// TwinCAT 3 PLC project PLC
// ProgramVersion: 3.1.4026.19
// libraries:
//   Tc2_DMX, * (Beckhoff Automation GmbH)
//   Tc2_Standard, * (Beckhoff Automation GmbH)
//   Tc2_System, * (Beckhoff Automation GmbH)
// project tree:
//   DUTs/ ENUM_InternalControl_StateMachine.TcDUT
//   GVLs/ GVL_DMX.TcGVL
//   POUs/ FB_ModuleLEDs.TcPOU, P_TestModuleLEDs.TcPOU
//   / Task.TcTTO
// real-time tasks:
//   TASK Task: cycle T#10ms, priority 1, ADS port 350
// I/O:
//   DEVICE Device 1 (EtherCAT), AmsNetId 10.1.181.84.2.1
//     Term 6 (EK1200) [EK1200-5000 EtherCAT Power supply (2A E-Bus)]
//       Term 3 (EL1809) [EL1809 16Ch. Dig. Input 24V, 3ms]
//       Term 4 (EL1809) [EL1809 16Ch. Dig. Input 24V, 3ms]
//       Term 5 (EL2008) [EL2008 8Ch. Dig. Output 24V, 0.5A]
//       Term 7 (EL2008) [EL2008 8Ch. Dig. Output 24V, 0.5A]
//       Term 8 (EL6851) [EL6851 DMX Master]
//       Term 12 (EL9011) [EL9011 End Terminal]
//   DEVICE Device 4 (USB) (disabled)
//   DEVICE Device 5 (COM Port) (disabled)
// variable links:
//   Device 1 (EtherCAT) <-> Device 1 (EtherCAT)/Term 6 (EK1200)/Term 5 (EL2008)
//     Term 6 (EK1200)/Term 3 (EL1809)/Channel 1/Input <-> Channel 1/Output
//   PLC/PLC Instance <-> Device 1 (EtherCAT)/Term 6 (EK1200)/Term 8 (EL6851)
//     Task Inputs/GVL_DMX.stDMXInDataLine01/bCyclicTxDDisabled <-> DMX Status/Cyclic TxD disabled
//     Task Inputs/GVL_DMX.stDMXInDataLine01/bDefaultDataSent <-> DMX Status/Default data sent
//     Task Inputs/GVL_DMX.stDMXInDataLine01/bFrameSentToggle <-> DMX Status/Frame sent toggle
//     Task Inputs/GVL_DMX.stDMXInDataLine01/bReceiveToggle <-> DMX Status/Receive toggle
//     Task Inputs/GVL_DMX.stDMXInDataLine01/bTransmitAccepted <-> DMX Status/Transmit accepted
//     Task Inputs/GVL_DMX.stDMXInDataLine01/bTxPDOToggle <-> DMX Status/TxPDO Toggle
//     Task Inputs/GVL_DMX.stDMXInDataLine01/byStartCode <-> DMX Status/Start code
//     Task Inputs/GVL_DMX.stDMXInDataLine01/wChannelLength <-> DMX Status/Channel length
//     Task Outputs/GVL_DMX.stDMXOutDataLine01/arrData[100] <-> DMX Channel 65-128/Channel 100
//     Task Outputs/GVL_DMX.stDMXOutDataLine01/arrData[101] <-> DMX Channel 65-128/Channel 101
//     Task Outputs/GVL_DMX.stDMXOutDataLine01/arrData[102] <-> DMX Channel 65-128/Channel 102
//     Task Outputs/GVL_DMX.stDMXOutDataLine01/arrData[103] <-> DMX Channel 65-128/Channel 103
//     Task Outputs/GVL_DMX.stDMXOutDataLine01/arrData[104] <-> DMX Channel 65-128/Channel 104
//     Task Outputs/GVL_DMX.stDMXOutDataLine01/arrData[105] <-> DMX Channel 65-128/Channel 105
//     Task Outputs/GVL_DMX.stDMXOutDataLine01/arrData[106] <-> DMX Channel 65-128/Channel 106
//     Task Outputs/GVL_DMX.stDMXOutDataLine01/arrData[107] <-> DMX Channel 65-128/Channel 107
//     Task Outputs/GVL_DMX.stDMXOutDataLine01/arrData[108] <-> DMX Channel 65-128/Channel 108
//     Task Outputs/GVL_DMX.stDMXOutDataLine01/arrData[109] <-> DMX Channel 65-128/Channel 109
//     Task Outputs/GVL_DMX.stDMXOutDataLine01/arrData[10] <-> DMX Channel 1-64/Channel 10
//     Task Outputs/GVL_DMX.stDMXOutDataLine01/arrData[110] <-> DMX Channel 65-128/Channel 110
//     Task Outputs/GVL_DMX.stDMXOutDataLine01/arrData[111] <-> DMX Channel 65-128/Channel 111
//     Task Outputs/GVL_DMX.stDMXOutDataLine01/arrData[112] <-> DMX Channel 65-128/Channel 112
//     Task Outputs/GVL_DMX.stDMXOutDataLine01/arrData[113] <-> DMX Channel 65-128/Channel 113
//     Task Outputs/GVL_DMX.stDMXOutDataLine01/arrData[114] <-> DMX Channel 65-128/Channel 114
//     Task Outputs/GVL_DMX.stDMXOutDataLine01/arrData[115] <-> DMX Channel 65-128/Channel 115
//     Task Outputs/GVL_DMX.stDMXOutDataLine01/arrData[116] <-> DMX Channel 65-128/Channel 116
//     Task Outputs/GVL_DMX.stDMXOutDataLine01/arrData[117] <-> DMX Channel 65-128/Channel 117
//     Task Outputs/GVL_DMX.stDMXOutDataLine01/arrData[118] <-> DMX Channel 65-128/Channel 118
//     Task Outputs/GVL_DMX.stDMXOutDataLine01/arrData[119] <-> DMX Channel 65-128/Channel 119
//     Task Outputs/GVL_DMX.stDMXOutDataLine01/arrData[11] <-> DMX Channel 1-64/Channel 11
//     Task Outputs/GVL_DMX.stDMXOutDataLine01/arrData[120] <-> DMX Channel 65-128/Channel 120
//     Task Outputs/GVL_DMX.stDMXOutDataLine01/arrData[121] <-> DMX Channel 65-128/Channel 121
//     Task Outputs/GVL_DMX.stDMXOutDataLine01/arrData[122] <-> DMX Channel 65-128/Channel 122
//     Task Outputs/GVL_DMX.stDMXOutDataLine01/arrData[123] <-> DMX Channel 65-128/Channel 123
//     Task Outputs/GVL_DMX.stDMXOutDataLine01/arrData[124] <-> DMX Channel 65-128/Channel 124
//     Task Outputs/GVL_DMX.stDMXOutDataLine01/arrData[125] <-> DMX Channel 65-128/Channel 125
//     Task Outputs/GVL_DMX.stDMXOutDataLine01/arrData[126] <-> DMX Channel 65-128/Channel 126
//     Task Outputs/GVL_DMX.stDMXOutDataLine01/arrData[127] <-> DMX Channel 65-128/Channel 127
//     Task Outputs/GVL_DMX.stDMXOutDataLine01/arrData[128] <-> DMX Channel 65-128/Channel 128
//     Task Outputs/GVL_DMX.stDMXOutDataLine01/arrData[12] <-> DMX Channel 1-64/Channel 12
//     Task Outputs/GVL_DMX.stDMXOutDataLine01/arrData[13] <-> DMX Channel 1-64/Channel 13
//     Task Outputs/GVL_DMX.stDMXOutDataLine01/arrData[14] <-> DMX Channel 1-64/Channel 14
//     Task Outputs/GVL_DMX.stDMXOutDataLine01/arrData[15] <-> DMX Channel 1-64/Channel 15
//     Task Outputs/GVL_DMX.stDMXOutDataLine01/arrData[16] <-> DMX Channel 1-64/Channel 16
//     Task Outputs/GVL_DMX.stDMXOutDataLine01/arrData[17] <-> DMX Channel 1-64/Channel 17
//     Task Outputs/GVL_DMX.stDMXOutDataLine01/arrData[18] <-> DMX Channel 1-64/Channel 18
//     Task Outputs/GVL_DMX.stDMXOutDataLine01/arrData[19] <-> DMX Channel 1-64/Channel 19
//     Task Outputs/GVL_DMX.stDMXOutDataLine01/arrData[1] <-> DMX Channel 1-64/Channel 1
//     Task Outputs/GVL_DMX.stDMXOutDataLine01/arrData[20] <-> DMX Channel 1-64/Channel 20
//     Task Outputs/GVL_DMX.stDMXOutDataLine01/arrData[21] <-> DMX Channel 1-64/Channel 21
//     Task Outputs/GVL_DMX.stDMXOutDataLine01/arrData[22] <-> DMX Channel 1-64/Channel 22
//     Task Outputs/GVL_DMX.stDMXOutDataLine01/arrData[23] <-> DMX Channel 1-64/Channel 23
//     Task Outputs/GVL_DMX.stDMXOutDataLine01/arrData[24] <-> DMX Channel 1-64/Channel 24
//     Task Outputs/GVL_DMX.stDMXOutDataLine01/arrData[25] <-> DMX Channel 1-64/Channel 25
//     Task Outputs/GVL_DMX.stDMXOutDataLine01/arrData[26] <-> DMX Channel 1-64/Channel 26
//     Task Outputs/GVL_DMX.stDMXOutDataLine01/arrData[27] <-> DMX Channel 1-64/Channel 27
//     Task Outputs/GVL_DMX.stDMXOutDataLine01/arrData[28] <-> DMX Channel 1-64/Channel 28
//     Task Outputs/GVL_DMX.stDMXOutDataLine01/arrData[29] <-> DMX Channel 1-64/Channel 29
//     Task Outputs/GVL_DMX.stDMXOutDataLine01/arrData[2] <-> DMX Channel 1-64/Channel 2
//     Task Outputs/GVL_DMX.stDMXOutDataLine01/arrData[30] <-> DMX Channel 1-64/Channel 30
//     Task Outputs/GVL_DMX.stDMXOutDataLine01/arrData[31] <-> DMX Channel 1-64/Channel 31
//     Task Outputs/GVL_DMX.stDMXOutDataLine01/arrData[32] <-> DMX Channel 1-64/Channel 32
//     Task Outputs/GVL_DMX.stDMXOutDataLine01/arrData[33] <-> DMX Channel 1-64/Channel 33
//     Task Outputs/GVL_DMX.stDMXOutDataLine01/arrData[34] <-> DMX Channel 1-64/Channel 34
//     Task Outputs/GVL_DMX.stDMXOutDataLine01/arrData[35] <-> DMX Channel 1-64/Channel 35
//     Task Outputs/GVL_DMX.stDMXOutDataLine01/arrData[36] <-> DMX Channel 1-64/Channel 36
//     Task Outputs/GVL_DMX.stDMXOutDataLine01/arrData[37] <-> DMX Channel 1-64/Channel 37
//     Task Outputs/GVL_DMX.stDMXOutDataLine01/arrData[38] <-> DMX Channel 1-64/Channel 38
//     Task Outputs/GVL_DMX.stDMXOutDataLine01/arrData[39] <-> DMX Channel 1-64/Channel 39
//     Task Outputs/GVL_DMX.stDMXOutDataLine01/arrData[3] <-> DMX Channel 1-64/Channel 3
//     Task Outputs/GVL_DMX.stDMXOutDataLine01/arrData[40] <-> DMX Channel 1-64/Channel 40
//     Task Outputs/GVL_DMX.stDMXOutDataLine01/arrData[41] <-> DMX Channel 1-64/Channel 41
//     Task Outputs/GVL_DMX.stDMXOutDataLine01/arrData[42] <-> DMX Channel 1-64/Channel 42
//     Task Outputs/GVL_DMX.stDMXOutDataLine01/arrData[43] <-> DMX Channel 1-64/Channel 43
//     Task Outputs/GVL_DMX.stDMXOutDataLine01/arrData[44] <-> DMX Channel 1-64/Channel 44
//     Task Outputs/GVL_DMX.stDMXOutDataLine01/arrData[45] <-> DMX Channel 1-64/Channel 45
//     Task Outputs/GVL_DMX.stDMXOutDataLine01/arrData[46] <-> DMX Channel 1-64/Channel 46
//     Task Outputs/GVL_DMX.stDMXOutDataLine01/arrData[47] <-> DMX Channel 1-64/Channel 47
//     Task Outputs/GVL_DMX.stDMXOutDataLine01/arrData[48] <-> DMX Channel 1-64/Channel 48
//     Task Outputs/GVL_DMX.stDMXOutDataLine01/arrData[49] <-> DMX Channel 1-64/Channel 49
//     Task Outputs/GVL_DMX.stDMXOutDataLine01/arrData[4] <-> DMX Channel 1-64/Channel 4
//     Task Outputs/GVL_DMX.stDMXOutDataLine01/arrData[50] <-> DMX Channel 1-64/Channel 50
//     Task Outputs/GVL_DMX.stDMXOutDataLine01/arrData[51] <-> DMX Channel 1-64/Channel 51
//     Task Outputs/GVL_DMX.stDMXOutDataLine01/arrData[52] <-> DMX Channel 1-64/Channel 52
//     Task Outputs/GVL_DMX.stDMXOutDataLine01/arrData[53] <-> DMX Channel 1-64/Channel 53
//     Task Outputs/GVL_DMX.stDMXOutDataLine01/arrData[54] <-> DMX Channel 1-64/Channel 54
//     Task Outputs/GVL_DMX.stDMXOutDataLine01/arrData[55] <-> DMX Channel 1-64/Channel 55
//     Task Outputs/GVL_DMX.stDMXOutDataLine01/arrData[56] <-> DMX Channel 1-64/Channel 56
//     Task Outputs/GVL_DMX.stDMXOutDataLine01/arrData[57] <-> DMX Channel 1-64/Channel 57
//     Task Outputs/GVL_DMX.stDMXOutDataLine01/arrData[58] <-> DMX Channel 1-64/Channel 58
//     Task Outputs/GVL_DMX.stDMXOutDataLine01/arrData[59] <-> DMX Channel 1-64/Channel 59
//     Task Outputs/GVL_DMX.stDMXOutDataLine01/arrData[5] <-> DMX Channel 1-64/Channel 5
//     Task Outputs/GVL_DMX.stDMXOutDataLine01/arrData[60] <-> DMX Channel 1-64/Channel 60
//     Task Outputs/GVL_DMX.stDMXOutDataLine01/arrData[61] <-> DMX Channel 1-64/Channel 61
//     Task Outputs/GVL_DMX.stDMXOutDataLine01/arrData[62] <-> DMX Channel 1-64/Channel 62
//     Task Outputs/GVL_DMX.stDMXOutDataLine01/arrData[63] <-> DMX Channel 1-64/Channel 63
//     Task Outputs/GVL_DMX.stDMXOutDataLine01/arrData[64] <-> DMX Channel 1-64/Channel 64
//     Task Outputs/GVL_DMX.stDMXOutDataLine01/arrData[65] <-> DMX Channel 65-128/Channel 65
//     Task Outputs/GVL_DMX.stDMXOutDataLine01/arrData[66] <-> DMX Channel 65-128/Channel 66
//     Task Outputs/GVL_DMX.stDMXOutDataLine01/arrData[67] <-> DMX Channel 65-128/Channel 67
//     Task Outputs/GVL_DMX.stDMXOutDataLine01/arrData[68] <-> DMX Channel 65-128/Channel 68
//     Task Outputs/GVL_DMX.stDMXOutDataLine01/arrData[69] <-> DMX Channel 65-128/Channel 69
//     Task Outputs/GVL_DMX.stDMXOutDataLine01/arrData[6] <-> DMX Channel 1-64/Channel 6
//     Task Outputs/GVL_DMX.stDMXOutDataLine01/arrData[70] <-> DMX Channel 65-128/Channel 70
//     Task Outputs/GVL_DMX.stDMXOutDataLine01/arrData[71] <-> DMX Channel 65-128/Channel 71
//     Task Outputs/GVL_DMX.stDMXOutDataLine01/arrData[72] <-> DMX Channel 65-128/Channel 72
//     Task Outputs/GVL_DMX.stDMXOutDataLine01/arrData[73] <-> DMX Channel 65-128/Channel 73
//     Task Outputs/GVL_DMX.stDMXOutDataLine01/arrData[74] <-> DMX Channel 65-128/Channel 74
//     Task Outputs/GVL_DMX.stDMXOutDataLine01/arrData[75] <-> DMX Channel 65-128/Channel 75
//     Task Outputs/GVL_DMX.stDMXOutDataLine01/arrData[76] <-> DMX Channel 65-128/Channel 76
//     Task Outputs/GVL_DMX.stDMXOutDataLine01/arrData[77] <-> DMX Channel 65-128/Channel 77
//     Task Outputs/GVL_DMX.stDMXOutDataLine01/arrData[78] <-> DMX Channel 65-128/Channel 78
//     Task Outputs/GVL_DMX.stDMXOutDataLine01/arrData[79] <-> DMX Channel 65-128/Channel 79
//     Task Outputs/GVL_DMX.stDMXOutDataLine01/arrData[7] <-> DMX Channel 1-64/Channel 7
//     Task Outputs/GVL_DMX.stDMXOutDataLine01/arrData[80] <-> DMX Channel 65-128/Channel 80
//     Task Outputs/GVL_DMX.stDMXOutDataLine01/arrData[81] <-> DMX Channel 65-128/Channel 81
//     Task Outputs/GVL_DMX.stDMXOutDataLine01/arrData[82] <-> DMX Channel 65-128/Channel 82
//     Task Outputs/GVL_DMX.stDMXOutDataLine01/arrData[83] <-> DMX Channel 65-128/Channel 83
//     Task Outputs/GVL_DMX.stDMXOutDataLine01/arrData[84] <-> DMX Channel 65-128/Channel 84
//     Task Outputs/GVL_DMX.stDMXOutDataLine01/arrData[85] <-> DMX Channel 65-128/Channel 85
//     Task Outputs/GVL_DMX.stDMXOutDataLine01/arrData[86] <-> DMX Channel 65-128/Channel 86
//     Task Outputs/GVL_DMX.stDMXOutDataLine01/arrData[87] <-> DMX Channel 65-128/Channel 87
//     Task Outputs/GVL_DMX.stDMXOutDataLine01/arrData[88] <-> DMX Channel 65-128/Channel 88
//     Task Outputs/GVL_DMX.stDMXOutDataLine01/arrData[89] <-> DMX Channel 65-128/Channel 89
//     Task Outputs/GVL_DMX.stDMXOutDataLine01/arrData[8] <-> DMX Channel 1-64/Channel 8
//     Task Outputs/GVL_DMX.stDMXOutDataLine01/arrData[90] <-> DMX Channel 65-128/Channel 90
//     Task Outputs/GVL_DMX.stDMXOutDataLine01/arrData[91] <-> DMX Channel 65-128/Channel 91
//     Task Outputs/GVL_DMX.stDMXOutDataLine01/arrData[92] <-> DMX Channel 65-128/Channel 92
//     Task Outputs/GVL_DMX.stDMXOutDataLine01/arrData[93] <-> DMX Channel 65-128/Channel 93
//     Task Outputs/GVL_DMX.stDMXOutDataLine01/arrData[94] <-> DMX Channel 65-128/Channel 94
//     Task Outputs/GVL_DMX.stDMXOutDataLine01/arrData[95] <-> DMX Channel 65-128/Channel 95
//     Task Outputs/GVL_DMX.stDMXOutDataLine01/arrData[96] <-> DMX Channel 65-128/Channel 96
//     Task Outputs/GVL_DMX.stDMXOutDataLine01/arrData[97] <-> DMX Channel 65-128/Channel 97
//     Task Outputs/GVL_DMX.stDMXOutDataLine01/arrData[98] <-> DMX Channel 65-128/Channel 98
//     Task Outputs/GVL_DMX.stDMXOutDataLine01/arrData[99] <-> DMX Channel 65-128/Channel 99
//     Task Outputs/GVL_DMX.stDMXOutDataLine01/arrData[9] <-> DMX Channel 1-64/Channel 9
//     Task Outputs/GVL_DMX.stDMXOutDataLine01/bDisableCyclicTxD <-> DMX Control/Disable cyclic TxD
//     Task Outputs/GVL_DMX.stDMXOutDataLine01/bSendDefaultData <-> DMX Control/Send default data
//     Task Outputs/GVL_DMX.stDMXOutDataLine01/bTransmitRequest <-> DMX Control/Transmit request
//     Task Outputs/GVL_DMX.stDMXOutDataLine01/byStartCode <-> DMX Control/Start code
//     Task Outputs/GVL_DMX.stDMXOutDataLine01/wChannelLength <-> DMX Control/Channel length

CONFIGURATION PLC
    RESOURCE PLC ON TwinCAT3
        TASK Task(INTERVAL := T#10ms, PRIORITY := 1);
        PROGRAM P_TestModuleLEDs WITH Task : P_TestModuleLEDs;
    END_RESOURCE
END_CONFIGURATION

// ---- DUTs/ENUM_InternalControl_StateMachine.TcDUT
{attribute 'qualified_only'}
{attribute 'strict'}
{attribute 'to_string'}
TYPE ENUM_InternalControl_StateMachine :
(
	READY := 0, 
	STANDBY,
	RUN,
	FAULT
);
END_TYPE

// ---- GVLs/GVL_DMX.TcGVL
{attribute 'qualified_only'}
VAR_GLOBAL
	stDMXInDataLine01               AT %I*	:	ST_EL6851InData;
	stDMXOutDataLine01              AT %Q*	:	ST_EL6851OutData;
	stCommandBuffer01						:	ST_DMXCommandBuffer;
	arrDMXProcessData						:	ARRAY [1..512] OF BYTE;
	HMI_State : ENUM_InternalControl_StateMachine := ENUM_InternalControl_StateMachine.STANDBY;       // 0=INIT, 1=STANDBY, 2=RUN (charge)
END_VAR

// ---- POUs/P_TestModuleLEDs.TcPOU
PROGRAM P_TestModuleLEDs
VAR
    LEDsRGBColor : FB_ModuleLEDs();
	State		 : ENUM_InternalControl_StateMachine := ENUM_InternalControl_StateMachine.STANDBY;
END_VAR

IF GVL_DMX.HMI_State = ENUM_InternalControl_StateMachine.STANDBY THEN
	LEDsRGBColor(eStateLeds := ENUM_InternalControl_StateMachine.STANDBY);

ELSIF GVL_DMX.HMI_State = ENUM_InternalControl_StateMachine.READY THEN
	LEDsRGBColor(eStateLeds := ENUM_InternalControl_StateMachine.READY);

ELSIF GVL_DMX.HMI_State = ENUM_InternalControl_StateMachine.RUN THEN
	LEDsRGBColor(eStateLeds := ENUM_InternalControl_StateMachine.RUN);

ELSIF GVL_DMX.HMI_State = ENUM_InternalControl_StateMachine.FAULT THEN
	LEDsRGBColor(eStateLeds := ENUM_InternalControl_StateMachine.FAULT);
	
ELSE
	LEDsRGBColor(eStateLeds := ENUM_InternalControl_StateMachine.STANDBY);
	
END_IF

END_PROGRAM

// ---- POUs/FB_ModuleLEDs.TcPOU
FUNCTION_BLOCK FB_ModuleLEDs
VAR_INPUT
	eStateLeds : ENUM_InternalControl_StateMachine; // Input state as a word like 'init', 'standby', etc.
END_VAR

VAR
    nLEDsQuantity : INT := 50;
    fbEL6851Communication   : FB_EL6851Communication;
    
    // Charge effect variables (moved from method to FB level)
    nChargePosition     : INT := 0;
    nChargeCounter      : INT := 0;
    bChargeInitialized  : BOOL := FALSE;
END_VAR

// Keep DMX comunication alive
M_DMXComunication(bEL6851CommunicationEnable := TRUE);

// State machine: set state based on colorMode input
IF eStateLeds = ENUM_InternalControl_StateMachine.READY THEN
	M_StaticColorFunction(byRed := 0, byGreen := 0, byBlue :=255);
	
ELSIF eStateLeds = ENUM_InternalControl_StateMachine.STANDBY THEN
	M_BreathingColorFunction(byRed := 255, byGreen := 30, byBlue :=0, byStepSize :=1);
	
ELSIF eStateLeds = ENUM_InternalControl_StateMachine.RUN THEN
	M_ChargeEffect(byStaticLEDs := 27, byRed := 0, byGreen := 255, byBlue := 0);

ELSIF eStateLeds = ENUM_InternalControl_StateMachine.FAULT THEN
	M_BreathingColorFunction(byRed := 255, byGreen := 0, byBlue :=0, byStepSize :=1);
	
ELSE
    M_BreathingColorFunction(byRed := 255, byGreen := 30, byBlue :=0, byStepSize :=1);
	
END_IF

METHOD PRIVATE M_BreathingColorFunction : BOOL
VAR_INPUT
    byRed         : BYTE; // Red (0-255)
    byGreen       : BYTE; // Green (0-255)
    byBlue        : BYTE; // Blue (0-255)
    byStepSize    : BYTE; // Stepsize for brightness change minimum 1
END_VAR

VAR_INST
    byStatBrightness  : BYTE := 0;
    bStatDirectionUp  : BOOL := TRUE;
END_VAR

VAR
    dni                : DINT;
    dnChannelBase      : DINT;
    byActualRed        : BYTE;
    byActualGreen      : BYTE;
    byActualBlue       : BYTE;
    iClearIdx          : INT;
END_VAR
FOR iClearIdx := 1 TO 512 DO
    GVL_DMX.arrDMXProcessData[iClearIdx] := 0;
END_FOR;

IF bStatDirectionUp THEN
    IF byStatBrightness > (255 - byStepSize) THEN
        byStatBrightness := 255;
        bStatDirectionUp := FALSE;
    ELSE
        byStatBrightness := byStatBrightness + byStepSize;
    END_IF
ELSE
    IF byStatBrightness < byStepSize THEN
        byStatBrightness := 0;
        bStatDirectionUp := TRUE;
    ELSE
        byStatBrightness := byStatBrightness - byStepSize;
    END_IF
END_IF

byActualRed   := TO_BYTE( (TO_UDINT(byRed)   * TO_UDINT(byStatBrightness)) / 255 );
byActualGreen := TO_BYTE( (TO_UDINT(byGreen) * TO_UDINT(byStatBrightness)) / 255 );
byActualBlue  := TO_BYTE( (TO_UDINT(byBlue)  * TO_UDINT(byStatBrightness)) / 255 );

FOR dni := 1 TO nLEDsQuantity DO
    dnChannelBase := (dni - 1) * 3 + 1;
    
    IF (dnChannelBase + 2) <= 512 THEN  // Changed from UPPER_BOUND to explicit 512 check
        GVL_DMX.arrDMXProcessData[dnChannelBase]     := byActualRed;
        GVL_DMX.arrDMXProcessData[dnChannelBase + 1] := byActualGreen;
        GVL_DMX.arrDMXProcessData[dnChannelBase + 2] := byActualBlue;
    ELSE
        M_BreathingColorFunction := FALSE;
        RETURN;
    END_IF
END_FOR

M_BreathingColorFunction := TRUE;
END_METHOD

METHOD PRIVATE M_ChargeEffect : BOOL
VAR_INPUT
    byStaticLEDs    : BYTE;
    byRed           : BYTE;
    byGreen         : BYTE;
    byBlue          : BYTE;
END_VAR

VAR_INST
    nDropletPosition    : INT;
    nCounter            : INT := 0;
    bInitialized        : BOOL := FALSE;
END_VAR

VAR
    dni                 : DINT;
    dnChannelBase       : DINT;
    nOffStart           : INT;
    byBrightness        : BYTE;
    nDistance           : INT;
    nCurrentLED         : INT;
END_VAR
nOffStart := TO_INT(byStaticLEDs);

// Initialize droplet at the END of the strip
IF NOT bInitialized THEN
    nDropletPosition := (nLEDsQuantity - nOffStart - 1);
    bInitialized := TRUE;
END_IF

// Move droplet every 15 cycles BACKWARDS (towards static LEDs)
nCounter := nCounter + 1;
IF nCounter >= 10 THEN
    nCounter := 0;
    nDropletPosition := nDropletPosition - 1;  // REVERSED: subtract instead of add
    
    // Loop back to end when reaching static LEDs
    IF nDropletPosition < 0 THEN
        nDropletPosition := (nLEDsQuantity - nOffStart - 1);
    END_IF
END_IF

// Set LED colors with smooth trail
FOR dni := 1 TO nLEDsQuantity DO
    dnChannelBase := (dni - 1) * 3 + 1;
    
    IF (dnChannelBase + 2) <= UPPER_BOUND(GVL_DMX.arrDMXProcessData, 1) THEN
        
        // Static LEDs (always ON)
        IF dni <= TO_DINT(byStaticLEDs) THEN
            byBrightness := 255;
        
        // Moving droplet with trail in OFF section
        ELSIF dni > TO_DINT(byStaticLEDs) THEN
            nCurrentLED := TO_INT(dni) - nOffStart;
            nDistance := nCurrentLED - nDropletPosition;
            
            // Main droplet
            IF nDistance = 0 THEN
                byBrightness := 255;
            
            // Trail AHEAD of droplet (moving towards static LEDs)
            ELSIF nDistance = 1 THEN
                byBrightness := 180;  // 70% brightness
            ELSIF nDistance = 2 THEN
                byBrightness := 100;  // 40% brightness
            ELSIF nDistance = 3 THEN
                byBrightness := 40;   // 15% brightness
            
            // All others OFF
            ELSE
                byBrightness := 0;
            END_IF
        
        ELSE
            byBrightness := 0;
        END_IF
        
        // Apply brightness to color
        GVL_DMX.arrDMXProcessData[dnChannelBase]     := TO_BYTE((TO_UDINT(byRed) * TO_UDINT(byBrightness)) / 255);
        GVL_DMX.arrDMXProcessData[dnChannelBase + 1] := TO_BYTE((TO_UDINT(byGreen) * TO_UDINT(byBrightness)) / 255);
        GVL_DMX.arrDMXProcessData[dnChannelBase + 2] := TO_BYTE((TO_UDINT(byBlue) * TO_UDINT(byBrightness)) / 255);
        
    ELSE
        M_ChargeEffect := FALSE;
        RETURN;
    END_IF
END_FOR

M_ChargeEffect := TRUE;
END_METHOD

METHOD PRIVATE M_DMXComunication : BOOL
VAR_INPUT
	bEL6851CommunicationEnable : BOOL := FALSE;
END_VAR
// DMX communication
IF bEL6851CommunicationEnable = TRUE THEN
	fbEL6851Communication(
		wSourceManufacturerID := 16#42_41,
		dwSourceDeviceID := 16#12_13_14_15,
		bEnableSendingData := TRUE,
		bSetCycleMode := TRUE,
		bSendDefaultData := FALSE,
		uiDataLength := 512,
		dwOptions := 0,
		stEL6851InData := GVL_DMX.stDMXInDataLine01,
		stEL6851OutData := GVL_DMX.stDMXOutDataLine01,
		stCommandBuffer := GVL_DMX.stCommandBuffer01,
		arrProcessData := GVL_DMX.arrDMXProcessData
	);
END_IF
END_METHOD

METHOD PRIVATE M_StaticColorFunction : BOOL

VAR_INPUT
    byRed               : BYTE; // Red (0-255)
    byGreen             : BYTE; // Green (0-255)
    byBlue              : BYTE; // Blue (0-255)
END_VAR

VAR
	dni                   : DINT;       // Loop variable
    dnChannelBase        : DINT;       // Base channel for each LED
END_VAR
FOR dni := 1 TO nLEDsQuantity DO
    dnChannelBase := (dni - 1) * 3 + 1; // Calculate base channel for this LED (R channel)
    IF (dnChannelBase + 2) <= UPPER_BOUND(GVL_DMX.arrDMXProcessData, 1) THEN // Verify we're not exceeding the DMX array bounds
            GVL_DMX.arrDMXProcessData[dnChannelBase]     := byRed;
            GVL_DMX.arrDMXProcessData[dnChannelBase + 1] := byGreen;
            GVL_DMX.arrDMXProcessData[dnChannelBase + 2] := byBlue;
    END_IF
END_FOR
END_METHOD

END_FUNCTION_BLOCK
